FUNCTION_BLOCK Netw
  (* Standard: 61499-2 *)
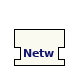
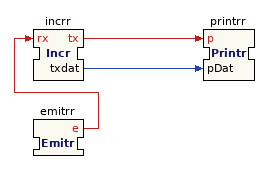
  FBS
    incrr : Incr;
    emitrr : Emitr;
    printrr : Printr;
  END_FBS
  EVENT_CONNECTIONS
    emitrr.e TO incrr.rx;
    incrr.tx TO printrr.p;
  END_CONNECTIONS
  DATA_CONNECTIONS
    incrr.txdat TO printrr.pDat;
  END_CONNECTIONS
END_FUNCTION_BLOCK
